// TIA Portal V16 export
// export: Created 2021-11-12T13:33:11.5256906Z, ExportSetting WithDefaults, DisplayName Totally Integrated Automation Portal, DisplayVersion V16 Update 3, DisplayName TIA Portal Version Control Interface, DisplayVersion V16 Update 2, DisplayName TIA Portal Openness, DisplayVersion V16 Update 3, DisplayName SINAMICS Startdrive Advanced, DisplayVersion V16 Update 5, DisplayName SINAMICS Startdrive G130, G150, S120, S150, SINAMICS MV, S210, DisplayVersion V16 Update 5, DisplayName SINAMICS Startdrive G110M, G120, G120C, G120D, G120P, G115D, DisplayVersion V16 Update 5, DisplayName STEP 7 Professional, DisplayVersion V16 Update 3, DisplayName STEP 7 Safety, DisplayVersion V16, DisplayName WinCC UA Professional, DisplayVersion V16 Update 3
DATA_BLOCK "IDB_Station450"   // DB197
VERSION : 0.1
// stored: AutoNumber true, DBAccessibleFromOPCUA true, InstanceOfName Station450, InstanceOfType FB
"Station450"
   // VAR
   //    SF_GL01_MA01 : "STD_Drive1";
   //    SF_GL02_MA01 { S7_SetPoint := 'True'} : "STD_Drive1";
   //    SF_GL03_MA01 { S7_SetPoint := 'True'} : "STD_Drive1";
   //    SF_GL04_MA01 { S7_SetPoint := 'True'} : "STD_Drive1";
   //    SF_UC21_TA1 { S7_SetPoint := 'True'} : "STD_Siemens_G120_CU240E_2_PN";
   //    SF_UC21_TA2 { S7_SetPoint := 'True'} : "STD_Siemens_G120_CU240E_2_PN";
   //    SF_UC21_TA3 { S7_SetPoint := 'True'} : "STD_Siemens_G120_CU240E_2_PN";
   //    SF_UC21_TA4 { S7_SetPoint := 'True'} : "STD_Siemens_G120_CU240E_2_PN";
   //    SF_BoxPartCounter { S7_SetPoint := 'True'} : "STD_PartCounter";
   //    SF_TON_BOX { S7_SetPoint := 'True'} : TON_TIME;
   //    SF_TOF_430TA01 { S7_SetPoint := 'True'} : TOF_TIME;
   //    SF_TOF_450TA01 { S7_SetPoint := 'True'} : TOF_TIME;
   //    SF_TOF_450TA02_1 { S7_SetPoint := 'True'} : TOF_TIME;
   //    SF_TOF_450TA02_2 { S7_SetPoint := 'True'} : TOF_TIME;
   //    SF_TOF_450TA04 { S7_SetPoint := 'True'} : TOF_TIME;
   //    SB1_PowerOk { S7_SetPoint := 'True'} : Bool;
   //    SB1BoxExchangeReq : Bool;
   //    SF_CL01_Alarm { S7_SetPoint := 'True'} : "STD_DI_Mon";
   //    SF_CL01_Warning { S7_SetPoint := 'True'} : "STD_DI_Mon";
   // END_VAR
BEGIN
END_DATA_BLOCK
